// SIMATIC S7-200 project (STEP 7-Micro/WIN), CPU 221 REL 01.10

SYMBOL_TABLE USER1
start            I0.0     // khoi dong he thong
estop            I0.1     // dung he thong
cb1              I0.2     // cam bien hop
cb2              I0.3     // cam bien tao
cb3              I0.4     // cong tac hanh trinh cua BTH
cb4              I0.5     // cong tac hanh trinh cua BTT
BTH              Q0.0     // Bang tai hop
BTT              Q0.1     // Bang tai tao
END_SYMBOL_TABLE

ORGANIZATION_BLOCK MAIN:OB1
TITLE=PROGRAM COMMENTS
BEGIN
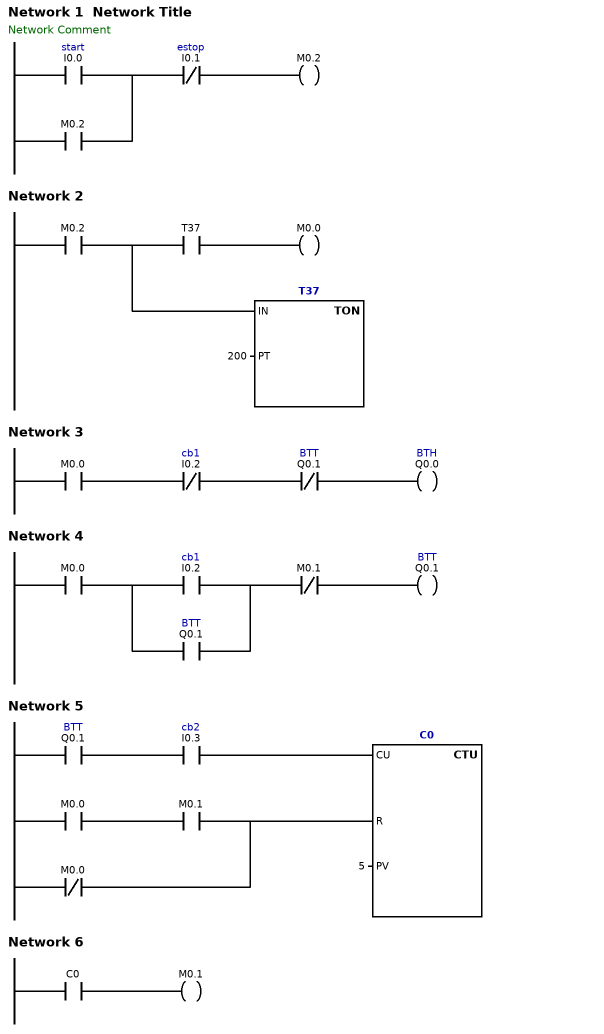
Network 1 // Network Title
// Network Comment
LD     start:I0.0
O      M0.2
AN     estop:I0.1
=      M0.2
Network 2
LD     M0.2
LPS
A      T37
=      M0.0
LPP
TON    T37, 200
Network 3
LD     M0.0
AN     cb1:I0.2
AN     BTT:Q0.1
=      BTH:Q0.0
Network 4
LD     M0.0
LD     cb1:I0.2
O      BTT:Q0.1
ALD
AN     M0.1
=      BTT:Q0.1
Network 5
LD     BTT:Q0.1
A      cb2:I0.3
LD     M0.0
A      M0.1
ON     M0.0
CTU    C0, 5
Network 6
LD     C0
=      M0.1
END_ORGANIZATION_BLOCK
